{attribute 'GeneratedUsingTerminal: EK1122-0000-0018'}
{attribute addProperty BoxType "EK1122-0000-0018"}
{attribute addProperty Id "Beckhoff_EM2xxxsub_EK1100EK1100_AB5A94672"}
{attribute addProperty CRC "1509611511"}
{attribute addProperty Size "2"}
TYPE Beckhoff_EM2xxxEK1122_59FAD7F7 EXTENDS EK1122_AB5A9467 :
STRUCT
	{attribute addProperty Name "Beckhoff_EM2xxxsub_EK1100"}
	Beckhoff_EM2xxxsub_EK1100 : EK1100_AB5A9467;
END_STRUCT
END_TYPE

(* stored: Version 1.2.0.0, ProductVersion 3.1.4024.9
   DUT Beckhoff_EM2xxxEK1122_59FAD7F7: Id {c9a0ba37-81de-4be6-8ae3-d90eceb65446} *)
